(* Schneider Machine Expert - Basic project automatic-water-bottle-filling-system, file version 2.7.0.0 *)
(* ProjectInformations: Name=New project *)

HARDWARE
  Cpu 0: TM221M16R/G
  EthernetConfiguration: NetworkName=M221, IpAllocationMode=FixedAddress, IpAddress=0.0.0.0, SubnetMask=0.0.0.0
  SerialLineConfiguration: Baud=Baud19200, Parity=ParityEven, DataBits=DataBits8, StopBits=StopBits1, PhysicalMedium=PhysicalMediumRs485, TransmissionMode=TransmissionModeModbusRtu, SlaveId=1, Addressing=SlaveAddressing
  MastTask: UsePeriodScanMode=false, PeriodScan=100
  FastTask: Period=255
  CpuBehavior: StartingMode=StartAsPreviousState, AutoSaveRamOnEeprom=true, WatchdogPeriod=250

SYMBOLS  (address, symbol, comment, settings)
  %I0.0     STARTED
  %I0.1     STOP
  %I0.2     IS_BOTTLE
  %I0.3     IS_FULL
  %Q0.0     CONVERYOR
  %Q0.1     VALVE

POU New POU
  (* SectionNumber=1 *)

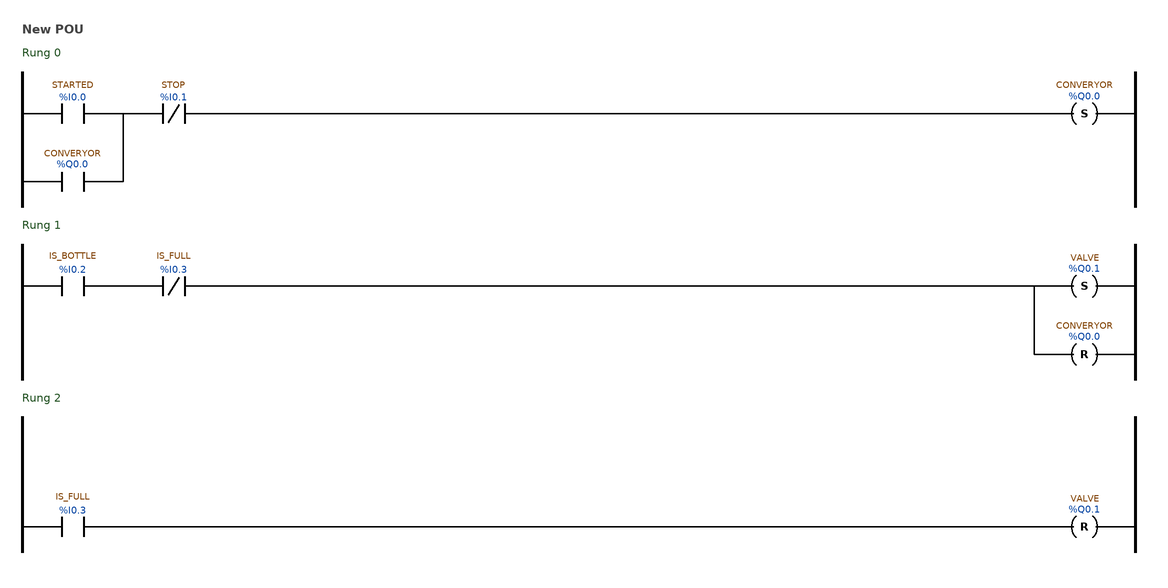

// Rung 0
  LD %I0.0                (* STARTED *)
  OR %Q0.0                (* CONVERYOR *)
  ANDN %I0.1              (* STOP *)
  S %Q0.0                 (* CONVERYOR *)
  // as ST:
  //   IF (STARTED OR CONVERYOR) AND NOT STOP THEN CONVERYOR := TRUE; END_IF;

// Rung 1
  LD %I0.2                (* IS_BOTTLE *)
  ANDN %I0.3              (* IS_FULL *)
  S %Q0.1                 (* VALVE *)
  R %Q0.0                 (* CONVERYOR *)
  // as ST:
  //   IF IS_BOTTLE AND NOT IS_FULL THEN VALVE := TRUE; END_IF;
  //   IF IS_BOTTLE AND NOT IS_FULL THEN CONVERYOR := FALSE; END_IF;

// Rung 2
  LD %I0.3                (* IS_FULL *)
  R %Q0.1                 (* VALVE *)
  // as ST:
  //   IF IS_FULL THEN VALVE := FALSE; END_IF;
